FUNCTION_BLOCK FB_LocalTest
VAR_INPUT
	fTime : LREAL;
	bEnableTest : BOOL;
END_VAR
VAR_OUTPUT
	fSignal : LREAL;
END_VAR
VAR
	fTempSignal : LREAL;
END_VAR

IF bEnableTest THEN
	fTempSignal := SIN(0.1 * 2 * Tc2_System.Global_Variables.PI * fTime);
	IF fTempSignal > 1.0 THEN
		fSignal := 1.0;
	ELSIF fTempSignal < -1.0 THEN
		fSignal := -1.0;
	ELSE
		fSignal := fTempSignal;
	END_IF
ELSE
	fTempSignal := 0.0;
END_IF

END_FUNCTION_BLOCK

(* stored: Version 1.1.0.1
   POU FB_LocalTest: Id {ab35aa25-2060-42c1-93b6-769f7cccc26b}, SpecialFunc None *)
